TYPE E_TcMatSimDataAreaType_1 :
(
	NotSpecified := 0,
	Standard,
	InputSrc,
	InputDst,
	OutputSrc,
	OutputDst,
	InternalDa,
	MArea,
	RetainDa
);
END_TYPE

(* stored: Version 1.1.0.1, ProductVersion 3.1.4020.12
   DUT E_TcMatSimDataAreaType_1: Id {2a3103c9-54a3-44c0-8cbe-1903edccf039} *)
